// Mitsubishi GX Works2 project: 기말과제 종근   PLC: Q02/Q02H
// 기기말과ㅘ제

PROGRAM MAIN
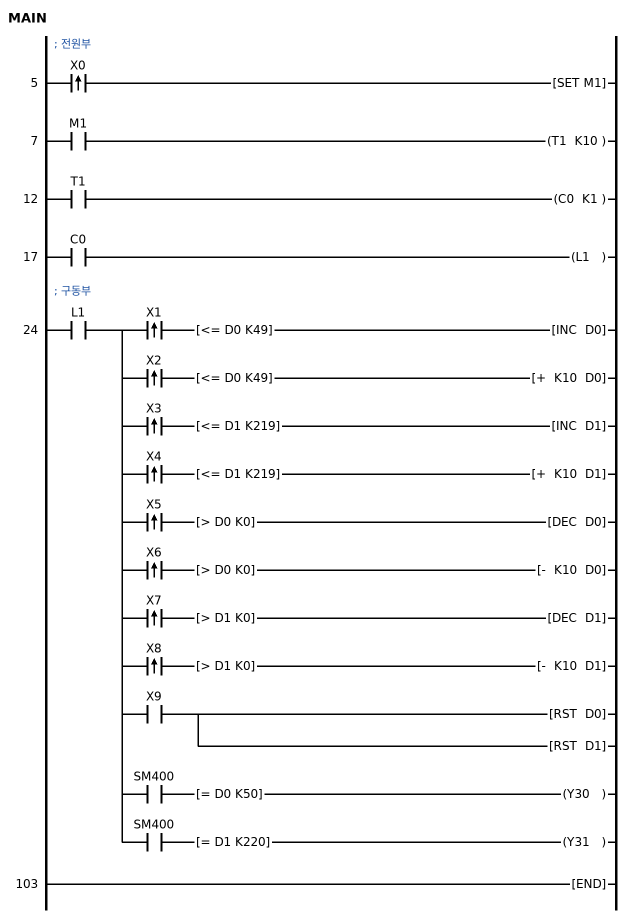
; 전원부
5     LDP     X0
      SET     M1
7     LD      M1
      OUT     T1 K10
12    LD      T1
      OUT     C0 K1
17    LD      C0
      OUT     L1
; 구동부
24    LD      L1
      MPS
      ANDP    X1
      AND<=   D0 K49
      INC     D0
      MRD
      ANDP    X2
      AND<=   D0 K49
      +       K10 D0
      MRD
      ANDP    X3
      AND<=   D1 K219
      INC     D1
      MRD
      ANDP    X4
      AND<=   D1 K219
      +       K10 D1
      MRD
      ANDP    X5
      AND>    D0 K0
      DEC     D0
      MRD
      ANDP    X6
      AND>    D0 K0
      -       K10 D0
      MRD
      ANDP    X7
      AND>    D1 K0
      DEC     D1
      MRD
      ANDP    X8
      AND>    D1 K0
      -       K10 D1
      MRD
      AND     X9
      RST     D0
      RST     D1
      MRD
      AND     SM400
      AND=    D0 K50
      OUT     Y30
      MPP
      AND     SM400
      AND=    D1 K220
      OUT     Y31
103   END
END_PROGRAM
